// TIA Portal V18 export
FUNCTION_BLOCK "fbSpeedControl"   // FB2, LAD
// stored: MemoryReserve 100, Namespace nsPerceuse, SetENOAutomatically false
   VAR_INPUT
      iFaster : Bool;
      iSlower : Bool;
   END_VAR
   VAR_IN_OUT
      ioSpeed : UDInt;
   END_VAR
BEGIN

REGION Network 1
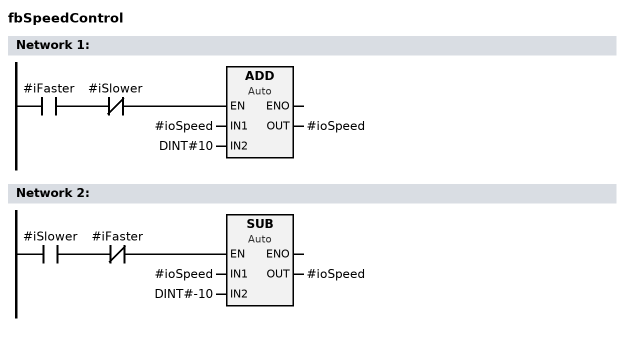
   RUNG wire#powerrail
      Contact( #iFaster )
      I_Contact( #iSlower )
      Add(in1 := #ioSpeed, in2 := DINT#10, out => #ioSpeed)
   END_RUNG
   // the same network as SCL:
   IF #iFaster AND NOT #iSlower THEN #ioSpeed := #ioSpeed + DINT#10; END_IF;
END_REGION

REGION Network 2
   RUNG wire#powerrail
      Contact( #iSlower )
      I_Contact( #iFaster )
      Sub(in1 := #ioSpeed, in2 := DINT#-10, out => #ioSpeed)
   END_RUNG
   // the same network as SCL:
   IF #iSlower AND NOT #iFaster THEN #ioSpeed := #ioSpeed - DINT#-10; END_IF;
END_REGION
END_FUNCTION_BLOCK
